FUNCTION_BLOCK Dose EXTENDS BaseState
VAR_INPUT
END_VAR
VAR_OUTPUT
END_VAR
VAR
END_VAR

METHOD mIrun : BOOL
FOR INDEX:=1 TO BasePointer^.pNUM_SILOS BY 1 DO
	IF BasePointer^.SiloFlagsAccessI[INDEX].pBufferedWeight - BasePointer^.LoadCellOutput[INDEX].ScaledValue >= BasePointer^.SiloFlagsAccessI[INDEX].pTargetWeight THEN
		BasePointer^.SpiralAccessI[INDEX].mAutoOff();
	END_IF
END_FOR

IF mCheckDosing() = TRUE THEN
	BasePointer^.MachineFlagsAccessI.pDosing := FALSE;
	ELSE
		RETURN;
END_IF

mNextState();
END_METHOD

END_FUNCTION_BLOCK

(* stored: Version 1.1.0.1, ProductVersion 3.1.4024.12
   POU Dose: Id {8405d10d-04a9-46b9-8c78-5923b7eebde8}, SpecialFunc None
   Method mIrun: Id {c11768bf-33f0-4646-8168-4155e99f20eb} *)
